# EPICS substitutions: iocs/MC08/tpmacApp/Db/pmacStatus.substitutions
file "db/pmacStatus.db"
{
pattern
{SYS,             PMAC,    VERSION  PLC  PORT,  NAXES }
{"XF:06BMA-BI",   "MC:08", "1",     5,   "P0",  8     }
}
